// TIA Portal V19 export
FUNCTION_BLOCK "S_Filter"   // FB18, LAD
TITLE = Sensor ON - OFF Filter
// stored: Access Published, MemoryReserve 100, SetENOAutomatically false
   VAR_INPUT
      S : Bool;
      PT_ON : Time;
      PT_OFF : Time;
   END_VAR
   VAR_IN_OUT
      S_F : Bool;
   END_VAR
   VAR
      TON_S_ON : TON_TIME;
      TON_S_OFF : TON_TIME;
   END_VAR
BEGIN

REGION Network 1: Exe
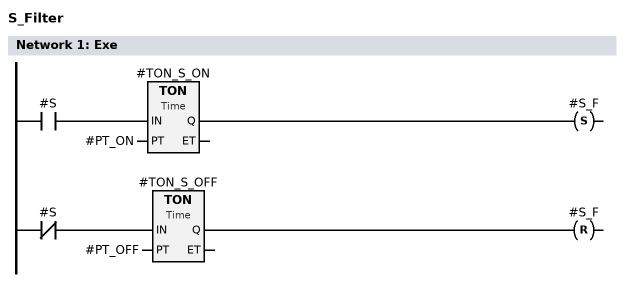
   RUNG wire#powerrail
      Contact( #S )
      { S7_Templates := "time_type := Time" } #TON_S_ON.TON(pt := #PT_ON, et =>)
      S_Coil( #S_F )
   END_RUNG
   RUNG wire#powerrail
      I_Contact( #S )
      { S7_Templates := "time_type := Time" } #TON_S_OFF.TON(pt := #PT_OFF, et =>)
      R_Coil( #S_F )
   END_RUNG
   // the same network as SCL:
   #TON_S_ON(IN := #S, PT := #PT_ON);   // TON
   IF #TON_S_ON.Q THEN #S_F := TRUE; END_IF;
   #TON_S_OFF(IN := NOT #S, PT := #PT_OFF);   // TON
   IF #TON_S_OFF.Q THEN #S_F := FALSE; END_IF;
END_REGION
END_FUNCTION_BLOCK
